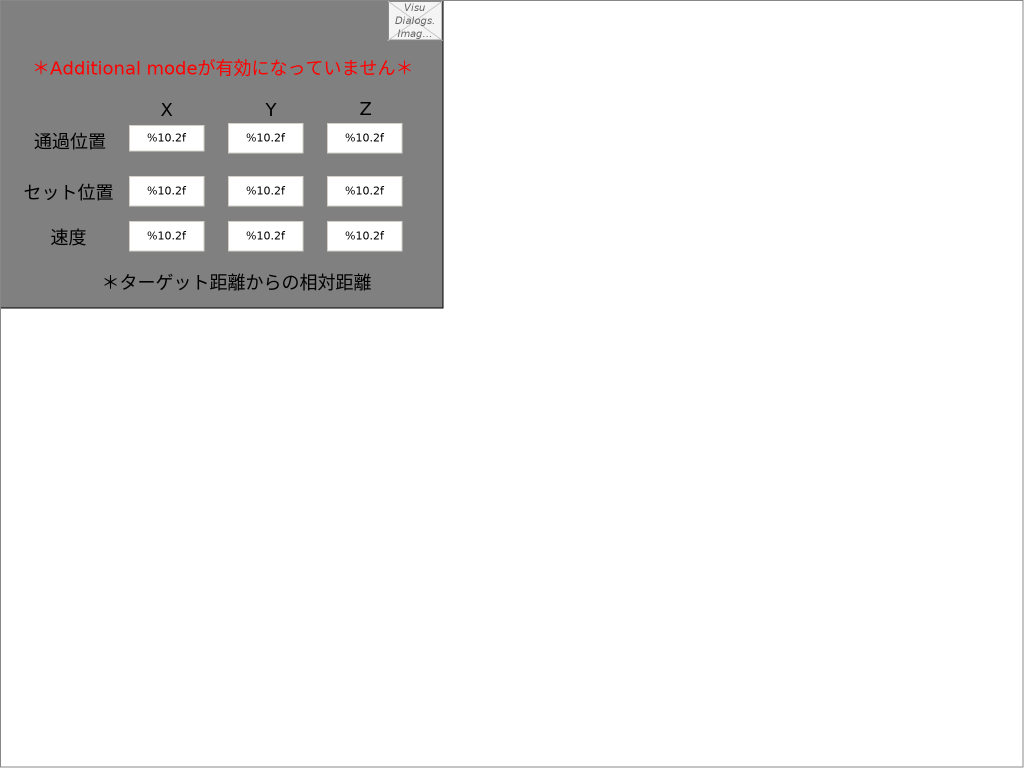
VISUALIZATION d_teahingDetail  // 1024x768
    Rectangle (0,0 443x308)
    Textfield (129,125 75x26), "%10.2f", text variable: gvl_visu.var_in_teachingDetail.passingPos.x
        OnMouseClick: write gvl_visu.var_in_teachingDetail.passingPos.x via VisuDialogs.Numpad, min -5, max 5
    Textfield (129,176 75x30), "%10.2f", text variable: gvl_visu.var_in_teachingDetail.settingPos.x
        OnMouseClick: write gvl_visu.var_in_teachingDetail.settingPos.x via VisuDialogs.Numpad, min -5, max 5
    Textfield (228,123 75x30), "%10.2f", text variable: gvl_visu.var_in_teachingDetail.passingPos.y
        OnMouseClick: write gvl_visu.var_in_teachingDetail.passingPos.y via VisuDialogs.Numpad, min -5, max 5
    Textfield (327,123 75x30), "%10.2f", text variable: gvl_visu.var_in_teachingDetail.passingPos.z
        OnMouseClick: write gvl_visu.var_in_teachingDetail.passingPos.z via VisuDialogs.Numpad, min -5, max 5
    Textfield (228,176 75x30), "%10.2f", text variable: gvl_visu.var_in_teachingDetail.settingPos.y
        OnMouseClick: write gvl_visu.var_in_teachingDetail.settingPos.y via VisuDialogs.Numpad, min -5, max 5
    Textfield (327,176 75x30), "%10.2f", text variable: gvl_visu.var_in_teachingDetail.settingPos.z
        OnMouseClick: write gvl_visu.var_in_teachingDetail.settingPos.z via VisuDialogs.Numpad, min -5, max 5
    Image (388,1 54x39), image: VisuDialogs.ImagePoolDialogs.Delete
        OnMouseClick: CloseDialog Dialog=d_teahingDetail, Result=OK, NumpadKeypadSet=True
    Label (18,178 101x30), "セット位置"
    Label (19,127 102x30), "通過位置"
    Label (125,95 84x30), "X"
    Label (324,94 84x30), "Z"
    Label (229,95 84x30), "Y"
    Label (71,260 331x46), "＊ターゲット距離からの相対距離"
    Label (16,48 414x41), "＊Additional modeが有効になっていません＊", invisible if: gvl_visu.var_dev_palletizingMode
    Textfield (129,221 75x30), "%10.2f", text variable: gvl_visu.var_in_teachingDetailVels.x.vel
        OnMouseClick: write gvl_visu.var_in_teachingDetailVels.x.vel via VisuDialogs.Numpad
    Textfield (228,221 75x30), "%10.2f", text variable: gvl_visu.var_in_teachingDetailVels.y.vel
        OnMouseClick: write gvl_visu.var_in_teachingDetailVels.y.vel via VisuDialogs.Numpad
    Textfield (327,221 75x30), "%10.2f", text variable: gvl_visu.var_in_teachingDetailVels.z.vel
        OnMouseClick: write gvl_visu.var_in_teachingDetailVels.z.vel via VisuDialogs.Numpad
    Label (18,223 101x30), "速度"
END_VISUALIZATION

(* stored: Version 1.1.0.1, ProductVersion 3.1.4024.12
   Visu d_teahingDetail: Id {73801335-463c-435c-9499-eea4f1ebb602} *)
